KUKA KRL program: pos_sub_pos.src

&ACCESS RV
&REL 15
&PARAM DISKPATH = Program/DEF
DEFFCT E6POS pos_sub_pos (e1 :IN, e2 :IN )
E6POS e1, e2

e1 = INIT_E6POS(e1, E6POS_NULL)
e2 = INIT_E6POS(e2, E6POS_NULL)

e1.X = e1.X - e2.X
e1.Y = e1.Y - e2.Y
e1.Z = e1.Z - e2.Z
e1.A = e1.A - e2.A
e1.B = e1.B - e2.B
e1.C = e1.C - e2.C

RETURN e1

ENDFCT
